{attribute 'strict'}
TYPE E_RTCCameraMethodState :
(
	RTC_CAMERA_METHOD_SEND_COMMAND 			:= 0,
	RTC_CAMERA_METHOD_RECEIVE_RESPONSE 		:= 10
);
END_TYPE

(* stored: Version 1.1.0.1, ProductVersion 3.1.4024.9
   DUT E_RTCCameraMethodState: Id {604b1db0-2d6e-41fc-9ca7-c914928de928} *)
